FUNCTION_BLOCK fbDigitalIO
VAR
	ioBIT : REFERENCE TO BOOL;
END_VAR

METHOD FB_init : BOOL
VAR_INPUT
	bInitRetains : BOOL; // if TRUE, the retain variables are initialized (warm start / cold start)
	bInCopyCode : BOOL;  // if TRUE, the instance afterwards gets moved into the copy code (online change)
	ioBitRef : REFERENCE TO BOOL;
END_VAR
ioBIT := ioBitRef;
END_METHOD

METHOD PUBLIC Get : BOOL
Get := ioBIT;
END_METHOD

END_FUNCTION_BLOCK

(* stored: Version 1.1.0.1, ProductVersion 3.1.4024.15
   POU fbDigitalIO: Id {433371ee-99e4-4f7a-9218-ad1d7806c1c1}, SpecialFunc None
   Method FB_init: Id {ca0d2adf-3d96-4140-8a80-3dbd673e4e5a}
   Method Get: Id {4623445c-48c3-4383-845f-2df71f63edb0} *)
